// TIA Portal V19 export
TYPE "LAF_typeConstraintWorkstationEm3Parameters"
// stored: Access Published
   STRUCT
      cm1Axis112 : "LAF_typeAxisParameters";
      cm2Axis113 { S7_SetPoint := 'True'} : "LAF_typeAxisParameters";
      cm3Axis115 { S7_SetPoint := 'True'} : "LAF_typeAxisParameters";
      cm4Axis116 { S7_SetPoint := 'True'} : "LAF_typeAxisParameters";
   END_STRUCT;
END_TYPE
